(* PLC project Unnamed, Неизвестно Unnamed 1 *)
(* stored: creationDateTime 2024-04-13T14:11:39, modificationDateTime 2024-04-13T15:48:28 *)

PROGRAM OLIA_examle
  VAR
    TestVar AT %QW0 : INT := 0;
  END_VAR
  VAR
    CTU0 : CTU;
    TON0 : TON;
    TP0 : TP;
  END_VAR
  VAR  (* added by the conversion: wires and edge detectors of the diagram *)
    R_TRIG1 : R_TRIG;
  END_VAR

(* FBD diagram, written out as Structured Text *)
TP0(IN := TON0.Q XOR True, PT := T#1000ms);
TON0(IN := TP0.Q, PT := T#500ms);
R_TRIG1(CLK := TON0.Q);
CTU0(CU := R_TRIG1.Q, R := CTU0.Q, PV := 100);
TestVar := CTU0.CV;
END_PROGRAM

CONFIGURATION Config0
  RESOURCE Res0 ON PLC
    TASK task0(INTERVAL := T#20ms, PRIORITY := 0);
    PROGRAM instance0 WITH task0 : OLIA_examle;
  END_RESOURCE
END_CONFIGURATION
